(* CODESYS project SPT_Vision.library
   Company: Beckhoff Automation LLC
   DefaultNamespace: SPT_Vision
   Version: 3.0.2
   Placeholder: SPT Vision
   Title: SPT Vision

Project tree, tasks and I/O mapping:
  libraries: SPT Base Types, * (Beckhoff Automation LLC); SPT Event Logger, * (Beckhoff Automation LLC); Tc2_EtherCAT, * (Beckhoff Automation GmbH); Tc2_Standard, * (Beckhoff Automation GmbH); Tc2_System, * (Beckhoff Automation GmbH); Tc2_Utilities, * (Beckhoff Automation GmbH); Tc3_EventLogger, * (Beckhoff Automation GmbH); Tc3_JsonXml, * (Beckhoff Automation GmbH); Tc3_Module, * (Beckhoff Automation GmbH); Tc3_Vision, * (Beckhoff Automation GmbH)
  DUTs/
  GVLs/
  POUs/
  Project Information/
    function F_GetCompany [ST]
    function F_GetTitle [ST]
    function F_GetVersion [ST]
  Version/
    global variables Global_Version
  Vision/
    DUTs/
      data type ST_CameraReadWrite
    GVLs/
      global variables GVL_VisionColor
    HMI/
      data type ST_VisionBase_Command
      data type ST_VisionBase_Config
      data type ST_VisionBase_HMI
      data type ST_VisionBase_Status
    PLC Task/
      function block FB_PlcCameraBase [ST]: CreateEvents, CyclicLogic, GetResults, Reset, RunVision, TriggerImage
    VisionTask/
      VideoPlayback/
        function block FB_ImageToVideo [ST]: Busy, Error, ErrorID, InitComplete, CyclicLogic, Execute, OnAlarmRaised, SubscribedEvents, SubscribeEvents, UnsubscribeEvents, AddImage, Initialize, Reset, TriggerAlarmForVideoCapture, WriteImage, CameraName, FramesPerSecond, JsonAttribute, ReductionFactor, TimeAfterEvent, TimeBeforeEvent, VideoOutputDirectory
      function block FB_VisionCameraBase [ST]: ExposureAddress, GainAddress, CyclicLogic, HMICommunication, ProcessImage, ReadParamUDINT, SetParamUDINT
    global variables Parameters_Vision
  VISUs/
*)

// Vision/DUTs/ST_CameraReadWrite
TYPE ST_CameraReadWrite :
	(*CameraCommand consists of Camera parameter address in HEX(byte)
	AND the data TO be written TO that address in decimal (UDINT).*)
	STRUCT
		CamAddress : UDINT;
		CamData	   : UDINT;
		Valid	   : BOOL;
	END_STRUCT
END_TYPE

// Vision/HMI/ST_VisionBase_Command
TYPE ST_VisionBase_Command :
	STRUCT
		StartAquisition : BOOL;
		StopAquisition	: BOOL;
		Trigger			: BOOL;
	END_STRUCT
END_TYPE

// Vision/HMI/ST_VisionBase_Config
TYPE ST_VisionBase_Config :
	STRUCT
		Gain			  : UDINT;
		SetGain			  : BOOL;
		ReadGain		  : BOOL;
		ReadGainValue	  : UDINT;
		Exposure		  : UDINT;
		SetExposure		  : BOOL;
		ReadExposure	  : BOOL;
		ReadExposureValue : UDINT;
	END_STRUCT
END_TYPE

// Vision/HMI/ST_VisionBase_HMI
TYPE ST_VisionBase_HMI :
	STRUCT
		Config	: ST_VisionBase_Config;
		Command : ST_VisionBase_Command;
		Status	: ST_VisionBase_Status;
	END_STRUCT
END_TYPE

// Vision/HMI/ST_VisionBase_Status
 
TYPE ST_VisionBase_Status :
	STRUCT
		VisionRunning : BOOL;
		CameraState	  : ETcVnCameraState;
		ElementsFound : UDINT;
	END_STRUCT
END_TYPE

// Version/Global_Version
{attribute 'TcGenerated'}
{attribute 'no-analysis'}
{attribute 'linkalways'}
// This function has been automatically generated from the project information.
VAR_GLOBAL CONSTANT
	{attribute 'const_non_replaced'}
	stLibVersion_SPT_Vision : ST_LibVersion := (iMajor := 3, iMinor := 0, iBuild := 2, iRevision := 0, nFlags := 1, sVersion := '3.0.2');
END_VAR

// Vision/GVLs/GVL_VisionColor
{attribute 'qualified_only'}
{attribute 'strict'}
VAR_GLOBAL
	ColorWhite	 : TcVnVector4_LREAL := [255, 255, 255, 255];
	ColorBlack	 : TcVnVector4_LREAL := [0, 0, 0, 255];
	ColorGreen	 : TcVnVector4_LREAL := [0, 175, 0, 255];
	ColorBlue	 : TcVnVector4_LREAL := [0, 0, 255, 255];
	ColorRed	 : TcVnVector4_LREAL := [255, 0, 0, 255];
	ColorMagenta : TcVnVector4_LREAL := [255, 0, 255, 255];
END_VAR

// Vision/Parameters_Vision
{attribute 'qualified_only'}
VAR_GLOBAL CONSTANT
	MAX_RESULTS_BUFFER_BYTES		  : UDINT := 1000;
	MAX_NUMBER_IMAGES_2_VIDEO		  : UDINT := 200;
	MAX_FRAMES_PER_SECOND			  : UDINT := 20;
	MAX_PERCENT_ROUTER_MEM_FOR_BUFFER : UDINT := 50;
	ADS_PORT_FOR_IMAGE_TO_VIDEO		  : UINT := 26129;
END_VAR

// Project Information/F_GetCompany
// This function has been automatically generated from the project information.
{attribute 'signature_flag' := '1073741824'}
{attribute 'TcGenerated'}
{attribute 'no-analysis'}
FUNCTION F_GetCompany : WSTRING
VAR_INPUT
	
END_VAR

F_GetCompany := "Beckhoff Automation LLC";

END_FUNCTION

// Project Information/F_GetTitle
// This function has been automatically generated from the project information.
{attribute 'signature_flag' := '1073741824'}
{attribute 'TcGenerated'}
{attribute 'no-analysis'}
FUNCTION F_GetTitle : WSTRING
VAR_INPUT
	
END_VAR

F_GetTitle := "SPT Vision";

END_FUNCTION

// Project Information/F_GetVersion
// This function has been automatically generated from the project information.
{attribute 'signature_flag' := '1073741824'}
{attribute 'TcGenerated'}
{attribute 'no-analysis'}
FUNCTION F_GetVersion : ST_LibVersion
VAR_INPUT
	
END_VAR

F_GetVersion.iMajor := 3;
F_GetVersion.iMinor := 0;
F_GetVersion.iBuild := 2;
F_GetVersion.iRevision := 0;
F_GetVersion.sVersion := '3.0.2';
F_GetVersion.nFlags := 1;

END_FUNCTION

// Vision/PLC Task/FB_PlcCameraBase
FUNCTION_BLOCK FB_PlcCameraBase EXTENDS FB_ComponentBase
VAR
	//Outputs
	SoftwareTrigger AT %Q* : BOOL;
	_RunVision		AT %Q* : BOOL;
	_Reset			AT %Q* : BOOL;
	ResultsReceived AT %Q* : BOOL;

	//Inputs
	CameraState		 AT %I* : ETcVnCameraState;
	ResultsAvailable AT %I* : BOOL;
	NumberOfResults	 AT %I* : UDINT;
	Results			 AT %I* : ARRAY[1..Parameters_Vision.MAX_RESULTS_BUFFER_BYTES] OF BYTE;
	VisionError		 AT %I* : BOOL;
	VisionErrorID	 AT %I* : UDINT;
	VisionAlarms			: ARRAY[1..5] OF FB_TcAlarm;
END_VAR

//! @summary Initializes event function blocks using this components's name
METHOD PROTECTED CreateEvents

//! @description This method is called by <c>Initialize()</c> as required
SUPER^.CreateEvents();

F_CreateAllEventsInClass(Alarms		:= VisionAlarms,
						 ClassSize	:= SIZEOF(TC_EVENTS.VisionBaseAlarms),
						 pInitEvent := ADR(TC_EVENTS.VisionBaseAlarms.InitReferenceEvent),
						 Prefix		:= Name);
END_METHOD

//! @summary This method serves as the entry point for all underlying FB logic
METHOD PUBLIC CyclicLogic

//! @description This method should be called cyclically by descendant function blocks by invoking <c>SUPER^.CyclicLogic()</c>.  Alternatively, the contents of this method could be reimplemented entirely in which case a call to this method would not be necessary.
SUPER^.CyclicLogic();

// Monitor camera error here
IF VisionError AND NOT VisionAlarms[E_VisionBaseAlarms.CameraFault].bRaised THEN
	VisionAlarms[E_VisionBaseAlarms.CameraFault].Raise(0);
ELSIF NOT VisionError AND VisionAlarms[E_VisionBaseAlarms.CameraFault].bRaised THEN
	VisionAlarms[E_VisionBaseAlarms.CameraFault].Clear(0, 0);
END_IF

_Error := VisionAlarms[E_VisionBaseAlarms.CameraFault].bRaised;
IF _Error THEN
	_ErrorID := VisionErrorID;
//ELSE
//	_ErrorID := 0;
END_IF

_Busy := _RunVision;
END_METHOD

METHOD GetResults : BOOL
VAR_IN_OUT
	ResultArray : ARRAY[1..Parameters_Vision.MAX_RESULTS_BUFFER_BYTES] OF BYTE;
	Number		: UDINT;
END_VAR

VAR_INST
	ResultsAvailable_RTRIG : R_TRIG;
END_VAR
GetResults := FALSE;
ResultsAvailable_RTRIG(CLK := ResultsAvailable);
IF ResultsAvailable_RTRIG.Q THEN
	IF SIZEOF(ResultArray) < SIZEOF(Results) THEN
		MEMCPY(ADR(ResultArray), ADR(Results), SIZEOF(ResultArray));
	ELSE
		MEMCPY(ADR(ResultArray), ADR(Results), SIZEOF(Results));
	END_IF

	IF NumberOfResults * SIZEOF(Results) > SIZEOF(ResultArray) THEN
		; ///Handle alarm
	END_IF

	Number	   := NumberOfResults;
	GetResults := TRUE;
	ResultsReceived := TRUE;
ELSE
	ResultsReceived := FALSE;
END_IF
END_METHOD

//! @summary Clears error flags and error IDs for this component
METHOD PUBLIC Reset : BOOL
//Return the value from the base FB Reset()
Reset := SUPER^.Reset();

// Clear the Vision Alarms
F_ClearAllEventsInClass(Alarms:=VisionAlarms);

// Set the Error ID to 0
_ErrorID := 0;
END_METHOD

PROPERTY RunVision : BOOL
SET
_RunVision := RunVision;
SoftwareTrigger := false;
END_SET
END_PROPERTY

PROPERTY TriggerImage : BOOL
SET
SoftwareTrigger := TriggerImage;
END_SET
END_PROPERTY

END_FUNCTION_BLOCK

// Vision/VisionTask/VideoPlayback/FB_ImageToVideo
FUNCTION_BLOCK FB_ImageToVideo EXTENDS FB_ListenerBase2 IMPLEMENTS I_CyclicFB
VAR_INPUT
END_VAR

VAR_OUTPUT
END_VAR

VAR
	//Base FB
	_Busy	 : BOOL := TRUE;
	_Error	 : BOOL;
	_ErrorID : UDINT;

	//Cyclic FB
	_InitComplete : BOOL;
	SequenceState : INT;

	//Reset
	_Reset : BOOL;

	//EnableImagesToBuffer : BOOL;
	TriggerVideoCapture : BOOL;
	VideoCaptureState	: INT;

	// Ring Buffer information
	BufferImageRing	 : ARRAY[1..Parameters_Vision.MAX_NUMBER_IMAGES_2_VIDEO] OF ITcVnImage;
	BufferIndex		 : UINT := 1;
	CurrentBufferMax : UINT;

	//BufferImageSaveIndex	  : UINT;
	WriteImageWaitResult	  : BOOL;
	ipImageForVideoRingBuffer : ITcVnImage;
	ipImageToSave			  : ITcVnImage;
	WriteFileState			  : INT;
	sImageToSaveName		  : STRING;
	fbWriteImage			  : FB_VN_WriteImage;
	SysTimeAtFileWrite		  : ULINT;
	_fbEvent				  : FB_TcEvent;
	ipImageWork				  : ITcVnImage;

	//Video creation vars
	writeADS   : ADSWRITE;
	DoWrite	   : BOOL;
	DataIn	   : ARRAY[1..4] OF BYTE;
	DoRead	   : BOOL;
	JSONData   : T_MaxString;
	JsonWriter : FB_JsonSaxWriter;

	//filename vars
	sFileName1						: T_MaxString;
	TimeDateStamp					: T_MaxString;
	GetTimeZone						: FB_GetTimeZoneInformation;
	TimeZoneInfo					: ST_TimeZoneInformation;
	SystemTimeToTzSpecificLocalTime : FB_SystemTimeToTzSpecificLocalTime;

	//CameraPlusCameraID : STRING;

	//Json vars to send to the C# app
	JsonFileName	: T_MaxString;
	JsonImageSource : T_MaxString;

	//Properties to build image
	_VideoOutputDirectory : STRING;
	_FramesPerSecond	  : UINT;
	_CameraName			  : STRING;
	_JSONAttribute		  : T_MaxString;
	_ReductionFactor	  : LREAL;

	//Alarm data
	sJsonAttribute	 : STRING(10000);
	JSONFilter		 : FB_TcEventFilter;
	_Subscribe		 : BOOL := TRUE;
	_Unsubscribe	 : BOOL;
	_Subscribed		 : BOOL;
	MissedEventCount : UDINT;

	//Image count value
	ImageWriteCount : UINT;
	FirstImage		: BOOL;

	//Delay after alarm to wait then do work
	AfterEventDelay	  : TON;
	_TimeAfterEvent	  : TIME;
	_TimeBeforeEvent  : TIME;
	StopImageAdding	  : BOOL;
	VideoCaptureAlarm : ARRAY[1..2] OF FB_TcAlarm;

	//Calculation of Video length variables
	ImageMemory				 : LREAL;
	VideoLengthCalculated	 : LREAL;
	VideoAskedLength		 : LREAL;
	TooLongForBufferFPS		 : BOOL;
	TooLongForMemory		 : BOOL;
	ImageMemCheckSize		 : ULINT := 0;
	RouterMem				 : FB_GetRouterStatusInfo;
	RouterInfo				 : ST_TcRouterStatusInfo;
	CheckMemorySize			 : BOOL := TRUE;
	NumberOfFramesCalculated : ULINT;
	CheckConnection			 : BYTE := 1;
	Check3rdParty_TON		 : TON;
	Check3rdParyRunning		 : BOOL;
END_VAR

PROPERTY Busy : BOOL
GET
Busy := _Busy;
END_GET
END_PROPERTY

PROPERTY Error : BOOL
GET
Error := _Error;
END_GET
END_PROPERTY

PROPERTY ErrorID : UDINT
GET
ErrorID := _ErrorID;
END_GET
END_PROPERTY

PROPERTY InitComplete : BOOL
GET
InitComplete := _InitComplete;
END_GET
END_PROPERTY

METHOD PUBLIC CyclicLogic
VAR_INPUT
END_VAR

VAR
	hr				: HRESULT;
	tmpIndex		: UINT;
	systemTimeNow	: TIMESTRUCT;
	tmpString		: STRING;
	EventTimestamp1 : TimeStruct;
	EventTimestamp2 : TimeStruct;
	sDump			: STRING;
END_VAR

VAR_INST
	x : UINT;
END_VAR
IF NOT _InitComplete THEN
	_InitComplete := Initialize();
	RETURN;
END_IF

// Call the Listener Execute
Execute();

// Subscribe to the event logger to messages with the JSON Attribute
IF _Subscribe THEN
	_Subscribe := FALSE;
	JSONFilter.Clear().JsonAttribute.Value.EqualTo(_JSONAttribute); //define all events (messages and alarms) from this eventclass   
	hr := Subscribe2(JSONFilter);									//subscribe to retrieve defined events
	IF SUCCEEDED(hr) THEN
		_Subscribed := TRUE;
	END_IF
END_IF

IF _Unsubscribe THEN
	_Unsubscribe := FALSE;
	hr			 := Unsubscribe();
	IF SUCCEEDED(hr) THEN
		_Subscribed := FALSE;
	END_IF
END_IF

// This is the state engine for when an alarm occurs that needs a video
CASE VideoCaptureState OF
	0:
		IF TriggerVideoCapture THEN
			_Busy			  := TRUE;
			x				  := 1;
			VideoCaptureState := 10;
		END_IF

	10: //wait for delay time to capture images after event
		IF AfterEventDelay.Q THEN
			StopImageAdding	  := TRUE;
			VideoCaptureState := 15;
		END_IF

	15: //save images needed for video playback
		WriteImageWaitResult := TRUE;
		tmpIndex			 := BufferIndex + x - 1;
		IF tmpIndex > CurrentBufferMax THEN
			tmpIndex := tmpIndex - CurrentBufferMax;
		END_IF

		IF WriteImage(Index := x, BufferImageSaveNameIndex := TmpIndex) THEN
			x := x + 1;
		END_IF

		IF x > CurrentBufferMax THEN
			TriggerVideoCapture	 := FALSE;
			StopImageAdding		 := FALSE;
			VideoCaptureState	 := 20;
			WriteImageWaitResult := FALSE;
		END_IF

	20: //Build string paths and names

		// Time is UTC and we need it in local time zone. 
		EventTimestamp1 := FILETIME64_TO_SYSTEMTIME(_fbevent.nTimestamp);
		SystemTimeToTzSpecificLocalTime(in := EventTimestamp1, tzInfo := TimeZoneInfo, out => EventTimestamp2);
		TimeDateStamp := SYSTEMTIME_TO_STRING(EventTimestamp2);
		FindAndReplaceChar(ADR(TimeDateStamp),
						   ':',
						   '-',
						   ADR(TimeDateStamp),
						   SIZEOF(TimeDateStamp));

		FindAndSplitChar(sSeparatorChar	  := '.',
						 pSrcString		  := ADR(TimeDateStamp),
						 pLeftString	  := ADR(TimeDateStamp),
						 nLeftSize		  := SIZEOF(TimeDateStamp),
						 pRightString	  := ADR(sDump),
						 nRightSize		  := SIZEOF(sDump),
						 bSearchFromRight := FALSE);

		//FileName string creation
		JsonFileName := CONCAT(_VideoOutputDirectory, '\');
		JsonFileName := CONCAT(JsonFileName, _CameraName);
		JsonFileName := CONCAT(JsonFileName, '\');
		JsonFileName := CONCAT(JsonFileName, TimeDateStamp);
		JsonFileName := CONCAT(JsonFileName, '.mp4');

		//image source string creation
		JsonImageSource	  := CONCAT(_VideoOutputDirectory, '\');
		JsonImageSource	  := CONCAT(JsonImageSource, _CameraName);
		JsonImageSource	  := CONCAT(JsonImageSource, '\');
		JsonImageSource	  := CONCAT(JsonImageSource, 'images');
		VideoCaptureState := 30;

	30: //setup JSON pairs
		MEMSET(ADR(JSONData), 0, SIZEOF(JSONData));
		JsonWriter.ResetDocument();
		JsonWriter.StartObject();
		JsonWriter.AddKeyString('ImagePathSource', JsonImageSource);
		JsonWriter.AddKeyString('VideoFilename', JsonFileName);
		JsonWriter.AddKeyNumber('VideoFPS', _FramesPerSecond);

		//JsonWriter.AddKeyLreal('ImageReductionFactor', _ImageReductionFactor);
		JsonWriter.EndObject();
		JSONData		  := JsonWriter.GetDocument();
		VideoCaptureState := 40;

	40: //write JSON data
		DoWrite			  := TRUE;
		VideoCaptureState := 45;

	45:
		IF writeADS.BUSY AND NOT writeADS.ERR THEN
			VideoCaptureState := 50;
		ELSIF writeADS.ERR THEN
			_ErrorID		  := writeADS.ERRID;
			VideoCaptureState := 999;
		END_IF

	50: //wait for write to be done
		IF NOT writeADS.BUSY AND NOT writeADS.ERR THEN
			DoWrite			  := FALSE;
			VideoCaptureState := 60;
		ELSIF writeADS.ERR THEN
			_ErrorID		  := writeADS.ERRID;
			VideoCaptureState := 999;
		END_IF

	60: //extra scan
		VideoCaptureAlarm[E_VideoAlarm.Camera1Alarm].Clear(0, 0);
		_Busy			  := FALSE;
		VideoCaptureState := 0;

	999: //error handling
		VideoCaptureAlarm[E_VideoAlarm.Camera1Alarm].Clear(0, 0);
		VideoCaptureAlarm[E_VideoAlarm.ImageToVideoService].Raise(0);
		DoWrite			  := FALSE;
		_Busy			  := FALSE;
		_Error			  := TRUE;
		VideoCaptureState := 1000;

	1000:
		IF _Reset THEN
			_Error			  := FALSE;
			_ErrorID		  := 0;
			VideoCaptureState := 0;
			_Reset			  := FALSE;
		END_IF
END_CASE

writeADS(NETID	 := '',
		 PORT	 := Parameters_Vision.ADS_PORT_FOR_IMAGE_TO_VIDEO,
		 IDXGRP	 := 1,
		 IDXOFFS := 1,
		 WRITE	 := DoWrite,
		 LEN	 := TO_UDINT(LEN(JSONData)),
		 SRCADDR := ADR(JSONData),
		 TMOUT	 := T#10S);

AfterEventDelay(IN := VideoCaptureState = 10, PT := _TimeAfterEvent);

(* Calculations for checking the video FPS, TimeBefore + TimeAfter, And Parameter.Maxbuffer size while related to image size
	The parameters that can be adjusted
		1. FramesPerSecond
		2. Time Before Event
		3. Time Afeter Event
		4. MAX Number of Frames
		5. Reduction Factor
		
	Fixed Parameters
		1. The memmory - 50% of router memory (Parameter_Vision.MAX_PERCENT_ROUTER_MEM_FOR_BUFFER in %)	
*)

//Monitor the actual needed buffer size
CurrentBufferMax := TO_UINT((TO_LREAL(_TimeAfterEvent) + TO_LREAL(_TimeBeforeEvent)) / 1000.0 * TO_LREAL(_FramesPerSecond));
IF CurrentBufferMax > Parameters_Vision.MAX_NUMBER_IMAGES_2_VIDEO THEN
	CurrentBufferMax := TO_UINT(Parameters_Vision.MAX_NUMBER_IMAGES_2_VIDEO);
END_IF

// Calculated Video length from parameters
VideoLengthCalculated := Parameters_Vision.MAX_NUMBER_IMAGES_2_VIDEO * 1000 / _FramesPerSecond;
VideoAskedLength	  := TO_LREAL(_TimeAfterEvent + _TimeBeforeEvent);
IF VideoAskedLength > VideoLengthCalculated THEN
	TooLongForBufferFPS := TRUE;
ELSE
	TooLongForBufferFPS := FALSE;
END_IF

(* Check to see if enough memory for what is expected
   Get the index to last picture taken*)
tmpIndex := BufferIndex - 1;
IF tmpIndex < 1 THEN
	tmpIndex := CurrentBufferMax;
END_IF

//Get Image size
F_VN_ExportImageSize(ipImage := BufferImageRing[tmpIndex], ImageMemCheckSize, S_OK);
IF ImageMemCheckSize > 0 THEN
	NumberOfFramesCalculated :=
		TO_ULINT(TO_LREAL(RouterInfo.maxMem) * TO_LREAL(Parameters_Vision.MAX_PERCENT_ROUTER_MEM_FOR_BUFFER) / 100.0 / TO_LREAL(ImageMemCheckSize));
END_IF

// Is the size of the buffer Larger than that based on parameters than is given
IF NumberOfFramesCalculated < Parameters_Vision.MAX_NUMBER_IMAGES_2_VIDEO AND ImageMemCheckSize > 0 THEN
	TooLongForMemory := TRUE;
ELSE
	TooLongForMemory := FALSE;
END_IF

// Check if 3rd party app is connected to ADS 
Check3rdParty_TON(IN := VideoCaptureAlarm[E_VideoAlarm.ImageToVideoService].bRaised AND NOT Check3rdParyRunning, PT := T#60S);
IF VideoCaptureAlarm[E_VideoAlarm.ImageToVideoService].bRaised AND (Check3rdParty_TON.Q OR Check3rdParyRunning) THEN
	Check3rdParyRunning := TRUE;

	// Do an ADS write to C# App to see if it is running
	writeADS(PORT	 := Parameters_Vision.ADS_PORT_FOR_IMAGE_TO_VIDEO,
			 IDXGRP	 := 10,
			 IDXOFFS := 10,
			 LEN	 := SIZEOF(CheckConnection),
			 SRCADDR := ADR(CheckConnection),
			 WRITE	 := TRUE,
			 TMOUT	 := T#3S);

	IF NOT writeADS.BUSY THEN
		IF NOT writeADS.ERR THEN
			VideoCaptureAlarm[E_VideoAlarm.ImageToVideoService].Clear(0, 0);
		END_IF

		Check3rdParyRunning := FALSE;
	END_IF
END_IF
END_METHOD

METHOD Execute : HRESULT
VAR_INPUT
END_VAR
Execute := SUPER^.Execute();
END_METHOD

METHOD OnAlarmRaised : HRESULT
VAR_INPUT
	fbEvent : REFERENCE TO FB_TcEvent;
END_VAR

VAR 
	hr : HRESULT;
END_VAR
// This is where we actually do the work
IF NOT TriggerVideoCapture THEN
	TriggerVideoCapture := TRUE;
	ImageWriteCount := 1;
	hr					:= fbEvent.GetJsonAttribute(sJsonAttribute, SIZEOF(sJsonAttribute));
	_fbEvent:=fbevent;
ELSE
	MissedEventCount := MissedEventCount + 1;
END_IF

OnAlarmRaised := S_OK;
END_METHOD

PROPERTY SubscribedEvents : BOOL
GET
SubscribedEvents := _Subscribed;
END_GET
END_PROPERTY

PROPERTY SubscribeEvents : BOOL
SET
_Subscribe := SubscribeEvents;
END_SET
END_PROPERTY

PROPERTY UnsubscribeEvents : BOOL
SET
_Unsubscribe := UnsubscribeEvents;
END_SET
END_PROPERTY

METHOD AddImage
VAR_INPUT
	ipImageIn : ITcVnImage;
END_VAR

VAR
	hrWD1					 : HRESULT;
	tStop1					 : DINT := 20000;
	tRest1					 : DINT;
	hr						 : HRESULT;
	PixelFormat				 : TcVnPixelFormat;
	ImageInfo				 : TcVnImageInfo;
	ImagePixelFormatChannels : BYTE;
	ImageEffectivePixelSize	 : UINT;
	ImageInWidth			 : UDINT;
	ImageInHeight			 : UDINT;
	ImageSmallWidth			 : UDINT;
	ImageSmallHeight		 : UDINT;
END_VAR
IF NOT WriteImageWaitResult THEN
	hrWD1 := F_VN_StartRelWatchdog(tStop1, S_OK);

	// reduce the image if needed
	hr						 := F_VN_GetImageInfo(ipImage := ipImageIn, stImageInfo := ImageInfo, hrPrev := hr);
	ImagePixelFormatChannels := ImageInfo.stPixelFormat.nChannels;
	ImageEffectivePixelSize	 := ImageInfo.stPixelFormat.nElementSize;
	ImageInWidth			 := ImageInfo.nWidth;
	ImageInHeight			 := ImageInfo.nHeight;
	IF _ReductionFactor <> 1 THEN
		ImageSmallWidth	 := LREAL_TO_UDINT(UDINT_TO_LREAL(ImageInWidth) * _ReductionFactor);
		ImageSmallHeight := LREAL_TO_UDINT(UDINT_TO_LREAL(ImageInHeight) * _ReductionFactor);

		// Image Width and Height must be even for video conversion
		IF (ImageSmallWidth MOD 2) <> 0 THEN // Check if "Odd"
			ImageSmallWidth := ImageSmallWidth - 1;
		END_IF

		IF (ImageSmallHeight MOD 2) <> 0 THEN // Check if "Odd"
			ImageSmallHeight := ImageSmallHeight - 1;
		END_IF

		hr := F_VN_ResizeImage(ipImageIn,
							   ipImageWork,
							   ImageSmallWidth,
							   ImageSmallHeight,
							   1,
							   hr);
	ELSE
		hr := F_VN_CopyImage(ipImageIn, ipImageWork, hr);
	END_IF

	hr	:= F_VN_CopyImage(ipImageWork, BufferImageRing[BufferIndex], hr);
	hrWD1		:= F_VN_StopWatchdog(hrWD1, tRest => tRest1);
	BufferIndex := BufferIndex + 1;
	IF BufferIndex > CurrentBufferMax THEN
		BufferIndex := 1;
	END_IF
END_IF
END_METHOD

METHOD Initialize : BOOL
VAR_INPUT
END_VAR
CASE SequenceState OF
	// Get the Timezone
	0:
		GetTimeZone(sNetID	 := '',
					bExecute := TRUE,
					tTimeout := T#5S,
					tzInfo	 => TimeZoneInfo);

		IF NOT GetTimeZone.bBusy AND NOT GetTimeZone.bError THEN
			GetTimeZone(sNetID := '', bExecute := FALSE);
			SequenceState := 10;
		ELSIF GetTimeZone.bError THEN
			_Error		  := TRUE;
			_ErrorID	  := 16#FFFFFFFF;
			SequenceState := 10;
		END_IF

	// Get the router memory
	10:
		RouterMem(sNetId   := '',
				  bExecute := TRUE,
				  tTimeout := T#3S,
				  bBusy	   =>,
				  bError   =>,
				  nErrID   =>,
				  info	   => RouterInfo);

		IF NOT RouterMem.bBusy THEN
			RouterMem(sNetId := '', bExecute := FALSE);
			SequenceState := 20;
		END_IF

	// Create alarms
	20:
		VideoCaptureAlarm[E_VideoAlarm.Camera1Alarm].CreateEx(stEventEntry := TC_EVENTS.VideoAlarm.Camera1Alarm, bWithConfirmation := FALSE, ipSourceInfo := 0);
		VideoCaptureAlarm[E_VideoAlarm.Camera1Alarm].SetJsonAttribute(sJsonAttribute := _JSONAttribute);
		VideoCaptureAlarm[E_VideoAlarm.Camera1Alarm].ipArguments.AddString(value := _CameraName);
		VideoCaptureAlarm[E_VideoAlarm.ImageToVideoService].CreateEx(stEventEntry := TC_EVENTS.VideoAlarm.ImageToVideoService, bWithConfirmation := FALSE, ipSourceInfo := 0);
		SequenceState := 30;

	30:
		// Do an ADS write to C# App to see if it is running
		writeADS(NETID := '',
				 PORT	 := Parameters_Vision.ADS_PORT_FOR_IMAGE_TO_VIDEO,
				 IDXGRP	 := 10,
				 IDXOFFS := 10,
				 LEN	 := SIZEOF(CheckConnection),
				 SRCADDR := ADR(CheckConnection),
				 WRITE	 := TRUE,
				 TMOUT	 := T#20S);

		IF NOT writeADS.BUSY THEN
			IF writeADS.ERR THEN
				VideoCaptureAlarm[E_VideoAlarm.ImageToVideoService].Raise(0);
			END_IF

			SequenceState := 40;
		END_IF

	40:
		Initialize := TRUE;
END_CASE
END_METHOD

METHOD Reset
VAR_INPUT
END_VAR
IF _Error THEN
	_Reset := TRUE;
END_IF
END_METHOD

METHOD PUBLIC TriggerAlarmForVideoCapture
VAR_INPUT
END_VAR
IF NOT VideoCaptureAlarm[E_VideoAlarm.Camera1Alarm].bRaised THEN
	VideoCaptureAlarm[E_VideoAlarm.Camera1Alarm].Raise(0);
END_IF
END_METHOD

METHOD WriteImage : BOOL
VAR_INPUT
	BufferImageSaveNameIndex : UINT;
	Index					 : UINT;
END_VAR

VAR
	SysTimeAtImageSave : ULINT;
END_VAR
CASE WriteFileState OF
	0:
		sImageToSaveName := CONCAT(STR1 := _VideoOutputDirectory, '\');
		sImageToSaveName := CONCAT(STR1 := sImageToSaveName, _CameraName);
		sImageToSaveName := CONCAT(STR1 := sImageToSaveName, '\Images\Image');
		CASE Index OF // Add leading zeros to index number of image name
			0..9:
				sImageToSaveName := CONCAT(sImageToSaveName, '000');
				sImageToSaveName := CONCAT(sImageToSaveName, TO_STRING(Index));

			10..99:
				sImageToSaveName := CONCAT(sImageToSaveName, '00');
				sImageToSaveName := CONCAT(sImageToSaveName, TO_STRING(Index));

			100..999:
				sImageToSaveName := CONCAT(sImageToSaveName, '0');
				sImageToSaveName := CONCAT(sImageToSaveName, TO_STRING(Index));

		ELSE
			sImageToSaveName := CONCAT(sImageToSaveName, TO_STRING(Index));
		END_CASE;

		sImageToSaveName   := CONCAT(sImageToSaveName, '.png');
		ipImageToSave	   := BufferImageRing[BufferImageSaveNameIndex];
		///SysTimeAtImageSave := F_GetSystemTime();
		WriteFileState	   := 10;

	10:
		// sFilePath must contain the full path, image name and type
		fbWriteImage(ipImage   := ipImageToSave,
					 sFilePath := sImageToSaveName,
					 nTimeout  := T#500MS,
					 bWrite	   := TRUE);

		IF NOT fbWriteImage.bBusy AND NOT fbWriteImage.bError THEN
			fbWriteImage(sFilePath := sImageToSaveName, bWrite := FALSE);
			WriteFileState := 0;
			WriteImage	   := TRUE;
		ELSIF fbWriteImage.bError THEN
			fbWriteImage(sFilePath := sImageToSaveName, bWrite := FALSE);
			WriteFileState := 0;
		END_IF

ELSE
	WriteFileState := 0;
END_CASE
END_METHOD

PROPERTY CameraName : STRING
SET
_CameraName := CameraName;
END_SET
END_PROPERTY

PROPERTY FramesPerSecond : UINT
SET
_FramesPerSecond := FramesPerSecond;
END_SET
END_PROPERTY

PROPERTY JsonAttribute : T_MaxString
SET
_JSONAttribute := JsonAttribute;
END_SET
END_PROPERTY

PROPERTY ReductionFactor : LREAL
SET
_ReductionFactor := ReductionFactor;
END_SET
END_PROPERTY

PROPERTY TimeAfterEvent : TIME
SET
_TimeAfterEvent := TimeAfterEvent;
END_SET
END_PROPERTY

PROPERTY TimeBeforeEvent : TIME
SET
_TimeBeforeEvent := TimeBeforeEvent;
END_SET
END_PROPERTY

PROPERTY VideoOutputDirectory : STRING
SET
_VideoOutputDirectory := VideoOutputDirectory;
END_SET
END_PROPERTY

END_FUNCTION_BLOCK

// Vision/VisionTask/FB_VisionCameraBase
FUNCTION_BLOCK ABSTRACT FB_VisionCameraBase EXTENDS FB_ComponentBase
VAR
	// Vision Related
	hr		   : HRESULT;
	Camera	   : FB_VN_SimpleCameraControl;
	ipImageIn  : ITcVnImage;
	ImageCount : ULINT;

	//Inputs to Camera
	RunVision		AT %I* : BOOL;
	SoftwareTrigger AT %I* : BOOL;
	Reset			AT %I* : BOOL;
	ResultsReceived AT %I* : BOOL;

	//Outputs From Camera (Property)
	CameraState		 AT %Q* : ETcVnCameraState;
	ResultsAvailable AT %Q* : BOOL;
	NumberOfResults	 AT %Q* : UDINT;
	Results			 AT %Q* : ARRAY[1..Parameters_Vision.MAX_RESULTS_BUFFER_BYTES] OF BYTE;
	VisionError		 AT %Q* : BOOL;
	VisionErrorID	 AT %Q* : UDINT;

	//Read Write Data
	_ReadData		: BOOL;
	_ReadAddress	: UDINT;
	_WriteData		: BOOL;
	_WriteValue		: UDINT;
	_WriteAddress	: UDINT;
	_ReadDataResult : BOOL;
	_ReadDataValue	: UDINT;
	_ReadDataValid	: BOOL;
	_WriteDataDone	: BOOL;

	//Camera Addresses
	_ExposureAddress : UDINT; //Default is zero and checked when asked to write
	_GainAddress	 : UDINT;

	//Camera Parameter Read/Write Section ******************************************************************
	WriteCamera			  : FB_VN_WriteRegister_UDINT;
	ReadCamera			  : FB_VN_ReadRegister_UDINT;
	ReadValue			  : UDINT;
	ReadCamera_FTRIG	  : F_TRIG;
	ReadCameraError_RTRIG : R_TRIG;

	// Timing Statistics
	SysTimeAtImageArrive : ULINT; // system time units = 1 nS
	SysTimeAtTrigger	 : ULINT; // system time units = 1 nS
	SysTimeAfterProcess	 : ULINT; // system time units = 1 nS
	_ProcessTime		 : LREAL;
	_TriggerToImageTime	 : LREAL;
	_TotalTime			 : LREAL;

	//Read/Write params
	tmpCamParamRead		  : ST_CameraReadWrite;
	tmpCamReadData		  : ST_CameraReadWrite;
	ReadCameraData_RTRIG  : R_TRIG;
	WriteCameraData_RTRIG : R_TRIG;

	//Trigger support
	SoftwareTrigger_RTRIG : R_TRIG;
	HMI_Trigger			  : BOOL;

	//HMI
	VisionBase_HMI : ST_VisionBase_HMI;


END_VAR

PROPERTY ExposureAddress : UDINT
SET
_ExposureAddress := ExposureAddress;
END_SET
END_PROPERTY

PROPERTY GainAddress : UDINT
SET
_GainAddress := GainAddress;
END_SET
END_PROPERTY

METHOD PUBLIC CyclicLogic
SUPER^.CyclicLogic();

// Do the camera logic
CameraState := Camera.GetState();
CASE CameraState OF
	// Initializing States to get to opened
	TCVN_CS_INITIAL, TCVN_CS_INITIALIZING, TCVN_CS_INITIALIZED, TCVN_CS_OPENING:
		hr := Camera.StartAcquisition();
		IF CameraState = TCVN_CS_INITIALIZED THEN
			VisionError := FALSE;
		END_IF

	// In opened, continue if application asks to run
	TCVN_CS_OPENED:
		IF RunVision THEN
			hr := Camera.StartAcquisition();
		END_IF

	// Always call another StartAquisition when in that state
	TCVN_CS_STARTACQUISITION:
		hr := Camera.StartAcquisition();

	// Response to the Triggering is to TriggerImage again
	TCVN_CS_TRIGGERING:
		hr := Camera.TriggerImage();

	// Waiting for image or application asked to stop running
	TCVN_CS_ACQUIRING:
		hr := Camera.GetCurrentImage(ipImageIn);

		// Check if new Image was received
		IF SUCCEEDED(hr) AND ipImageIn <> 0 THEN
			ResultsAvailable := FALSE;
			SysTimeAtImageArrive := F_GetActualDcTime64(); // get system time at new image
			ImageCount			 := ImageCount + 1;
			ProcessImage();
			SysTimeAfterProcess := F_GetActualDcTime64();
			ResultsAvailable	:= TRUE;
			_ProcessTime		:= TO_LREAL(SysTimeAfterProcess - SysTimeAtImageArrive) / TO_LREAL(Tc2_EtherCAT.EC_DCTIME_TICKSPERMSEC64);
			_TriggerToImageTime := TO_LREAL(SysTimeAtImageArrive - SysTimeAtTrigger) / TO_LREAL(Tc2_EtherCAT.EC_DCTIME_TICKSPERMSEC64);
			_TotalTime			:= TO_LREAL(SysTimeAfterProcess - SysTimeAtTrigger) / TO_LREAL(Tc2_EtherCAT.EC_DCTIME_TICKSPERMSEC64);
		ELSIF NOT RunVision THEN
			Camera.StopAcquisition();
		END_IF

	// Stop acqusition requires another call to StopAcquisiton
	TCVN_CS_STOPACQUISITION:
		hr := Camera.StopAcquisition();

	///UH oh.  We are in an error state  try to reset and initialize
	TCVN_CS_ERROR:
		VisionError			:= TRUE;
		hr := Camera.Reset();
END_CASE

//Handle Triggering here
SoftwareTrigger_RTRIG(CLK := (SoftwareTrigger OR HMI_Trigger));
IF SoftwareTrigger_RTRIG.Q THEN
	ResultsAvailable := FALSE;
	hr				 := Camera.TriggerImage();
	IF SUCCEEDED(hr) THEN
		SysTimeAtTrigger := F_GetActualDcTime64();
	END_IF
END_IF

IF ResultsReceived THEN
	ResultsAvailable := FALSE;
END_IF

(* Read/Write Camera Data ****************************************************************************
 Check for data in Process Image*)
ReadCameraData_RTRIG(CLK := _ReadData);
IF ReadCameraData_RTRIG.Q THEN
	_ReadDataResult		:= FALSE;
	ReadCamera.nAddress := _ReadAddress;
	ReadCamera.bRead	:= TRUE;
END_IF

ReadCamera(nEndian := 0, nTimeout := T#5S);
ReadCameraError_RTRIG(Clk := ReadCamera.bError AND ReadCamera.bRead AND NOT ReadCamera.bBusy);
ReadCamera.bRead := FALSE;
ReadCamera_FTRIG(CLK := ReadCamera.bBusy);
IF ReadCamera_FTRIG.Q OR ReadCameraError_RTRIG.Q THEN
	IF ReadCamera.bError THEN //ADSERR_DEVICE_BUSY
		_ReadDataResult := TRUE;
		_ReadDataValid	:= FALSE;
	ELSE
		_ReadDataResult := TRUE;
		_ReadDataValue	:= ReadCamera.nValue;
		_ReadDataValid	:= TRUE;
	END_IF
END_IF

WriteCameraData_RTRIG(CLK := _WriteData);

// Check Queue of parameters and Write to Camera
IF WriteCameraData_RTRIG.Q THEN
	_WriteDataDone		 := FALSE;
	WriteCamera.nAddress := _WriteAddress;
	WriteCamera.nValue	 := _WriteValue;
	WriteCamera.bWrite	 := TRUE;
END_IF

WriteCamera(nEndian := 0, nTimeout := T#5S);
WriteCamera.bWrite := FALSE;
IF _WriteData AND (NOT WriteCamera.bBusy OR WriteCamera.bError) THEN
	_WriteDataDone := TRUE;
END_IF

HMICommunication();
END_METHOD

METHOD PROTECTED HMICommunication
VAR_INPUT
END_VAR

VAR_INST
	Trigger_RTRIG	   : R_TRIG;
	ReadExposure_RTRIG : R_TRIG;
	ReadGain_RTRIG	   : R_TRIG;
	SetExposure_RTRIG  : R_TRIG;
	SetGain_RTRIG	   : R_TRIG;
	ReadGain		   : BOOL;
	ReadExposure	   : BOOL;
	SetGain			   : BOOL;
	SetExposure		   : BOOL;
END_VAR
SUPER^.HMICommunication();

Trigger_RTRIG(CLK := VisionBase_HMI.Command.Trigger);
ReadExposure_RTRIG(CLK := VisionBase_HMI.Config.ReadExposure);
ReadGain_RTRIG(CLK := VisionBase_HMI.Config.ReadGain);
SetExposure_RTRIG(CLK := VisionBase_HMI.Config.SetExposure);
SetGain_RTRIG(CLK := VisionBase_HMI.Config.SetGain);

// handle the request to run vision
IF ComponentBase_HMI.Status.HMIControlAvailable THEN
	IF VisionBase_HMI.Command.StartAquisition THEN
		RunVision := TRUE;
	ELSIF VisionBase_HMI.Command.StopAquisition THEN
		RunVision := FALSE;
	END_IF

	IF ReadExposure_RTRIG.Q AND NOT _ReadData THEN
		ReadExposure := TRUE;
		_ReadAddress := _ExposureAddress;
		_ReadData	 := TRUE;
	ELSIF _ReadDataResult AND ReadExposure THEN
		_ReadData								:= FALSE;
		_ReadDataResult							:= FALSE;
		ReadExposure							:= FALSE;
		VisionBase_HMI.Config.ReadExposureValue := _ReadDataValue;
	END_IF

	IF ReadGain_RTRIG.Q AND NOT _ReadData THEN
		ReadGain	 := TRUE;
		_ReadAddress := _GainAddress;
		_ReadData	 := TRUE;
	ELSIF _ReadDataResult AND ReadGain THEN
		_ReadData							:= FALSE;
		_ReadDataResult						:= FALSE;
		ReadGain							:= FALSE;
		VisionBase_HMI.Config.ReadGainValue := _ReadDataValue;
	END_IF

	IF SetExposure_RTRIG.Q AND NOT _WriteData THEN
		_WriteData	  := TRUE;
		SetExposure	  := TRUE;
		_WriteAddress := _ExposureAddress;
		_WriteValue	  := VisionBase_HMI.Config.Exposure;
	ELSIF _WriteDataDone AND SetExposure THEN
		SetExposure	   := FALSE;
		_WriteDataDone := FALSE;
		_WriteData	   := FALSE;
	END_IF

	IF SetGain_RTRIG.Q AND NOT _WriteData THEN
		SetGain		  := TRUE;
		_WriteData	  := TRUE;
		_WriteAddress := _GainAddress;
		_WriteValue	  := VisionBase_HMI.Config.Gain;
	ELSIF _WriteDataDone AND SetGain THEN
		SetGain		   := FALSE;
		_WriteDataDone := FALSE;
		_WriteData	   := FALSE;
	END_IF

	HMI_Trigger := Trigger_RTRIG.Q;
ELSE
	_ReadData		:= FALSE;
	_ReadDataResult := FALSE;
END_IF

VisionBase_HMI.Status.VisionRunning := RunVision;
VisionBase_HMI.Status.CameraState	:= CameraState;
VisionBase_HMI.Status.ElementsFound := NumberOfResults;
END_METHOD

METHOD PUBLIC ABSTRACT ProcessImage
END_METHOD

METHOD PROTECTED ReadParamUDINT : BOOL
VAR_INPUT
	Address : UDINT;
END_VAR

VAR_IN_OUT
	Value : UDINT;
	Valid : BOOL;
END_VAR
ReadParamUDINT := FALSE;
IF NOT _ReadData THEN
	_ReadData := TRUE;
ELSIF _ReadDataResult THEN
	_ReadData		:= FALSE;
	_ReadDataResult := FALSE;
	Valid			:= _ReadDataValid;
	Value			:= _ReadDataValue;
	ReadParamUDINT	:= TRUE;
END_IF
END_METHOD

METHOD PROTECTED SetParamUDINT : BOOL
VAR_INPUT
	Value	: UDINT;
	Address : UDINT;
END_VAR
SetParamUDINT := FALSE;
IF NOT _WriteData THEN
	_WriteData := TRUE;
	_WriteAddress := Address;
	_WriteValue := Value;
ELSIF _WriteDataDone THEN
	_WriteDataDone := FALSE;
	_WriteData := FALSE;
	SetParamUDINT := TRUE;
END_IF
END_METHOD

END_FUNCTION_BLOCK
